PROGRAM Initialize_Measurement_Values
VAR
	n : INT:=1;
	c : INT;

END_VAR

// Setting PCB
// Measurement Types 
// CSQ | CSD | CSR | CPQ | CPD | CPR | CPG | LSQ |LSD | LSR |
// LPQ | LPD | LPR | LPG | ZTH | YTH | RX | GB | DCR |
IF n<9 THEN
	// Setting Measurement Point 1 Resistance1
	c:=1;
	GVL.PLC_Data[n].Measure_Type[c] 		:='RX';
	GVL.PLC_Data[n].Measure_Reference[c]	:=680;
	GVL.PLC_Data[n].Measure_Tolerance[c]	:=34;
	// Setting Measurement Point 2 Capacitance1
	c:=2;
	GVL.PLC_Data[n].Measure_Type[c] 		:='CPQ';
	GVL.PLC_Data[n].Measure_Reference[c]	:=2.2E-08;
	GVL.PLC_Data[n].Measure_Tolerance[c]	:=2.2E-09;
	// Setting Measurement Point 3 Resistance2
	c:=3;
	GVL.PLC_Data[n].Measure_Type[c] 		:='RX';
	GVL.PLC_Data[n].Measure_Reference[c]	:=680;
	GVL.PLC_Data[n].Measure_Tolerance[c]	:=34;
		// Setting Measurement Point 3 Inductor 2
	c:=4;
	GVL.PLC_Data[n].Measure_Type[c] 		:='LPD';
	GVL.PLC_Data[n].Measure_Reference[c]	:=5;
	GVL.PLC_Data[n].Measure_Tolerance[c]	:=10;
		// Setting Measurement Point 3 Resistor 1
	c:=5;
	GVL.PLC_Data[n].Measure_Type[c] 		:='LPD';
	GVL.PLC_Data[n].Measure_Reference[c]	:=5;
	GVL.PLC_Data[n].Measure_Tolerance[c]	:=10;
		// Setting Measurement Point 3 Resistor 2
	c:=6;
	GVL.PLC_Data[n].Measure_Type[c] 		:='LPD';
	GVL.PLC_Data[n].Measure_Reference[c]	:=5;
	GVL.PLC_Data[n].Measure_Tolerance[c]	:=10;


    n:=n+1;

IF n=9 THEN
	GVL.Measurement_Init:= TRUE;
END_IF

END_IF

END_PROGRAM

(* stored: Version 1.1.0.1, ProductVersion 3.1.4024.3
   POU Initialize_Measurement_Values: Id {3a933f0f-d742-4163-8291-2877737c9b10}, SpecialFunc None *)
